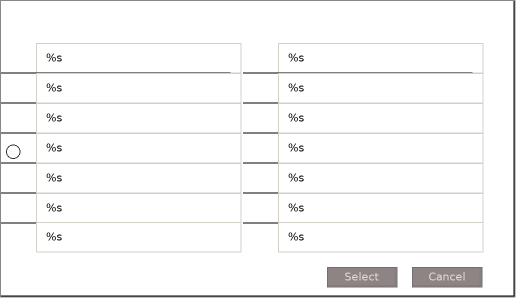
VISUALIZATION Visualization_FileList  // 516x298
    Rectangle (-1,0 515x296)
    Textfield (36,43 205x30), "%s", text variable: PRG_Process.arrFileNameList[1]
    Label (181,-2 158x39), "G-Code List"
    Line (230,73) (1,73)
    Line (230,103) (1,103)
    Line (230,133) (1,133)
    Line (230,163) (1,163)
    Line (230,193) (1,193)
    Line (230,223) (1,223)
    Textfield (36,73 205x30), "%s", text variable: PRG_Process.arrFileNameList[2]
    Textfield (36,103 205x30), "%s", text variable: PRG_Process.arrFileNameList[3]
    Textfield (36,133 205x30), "%s", text variable: PRG_Process.arrFileNameList[4]
    Textfield (36,163 205x30), "%s", text variable: PRG_Process.arrFileNameList[5]
    Textfield (36,193 205x30), "%s", text variable: PRG_Process.arrFileNameList[6]
    Textfield (36,222 205x30), "%s", text variable: PRG_Process.arrFileNameList[7]
    Textfield (278,43 205x30), "%s", text variable: PRG_Process.arrFileNameList[8]
    Line (472,73) (243,73)
    Line (472,103) (243,103)
    Line (472,133) (243,133)
    Line (472,163) (243,163)
    Line (472,193) (243,193)
    Line (472,223) (243,223)
    Textfield (278,73 205x30), "%s", text variable: PRG_Process.arrFileNameList[9]
    Textfield (278,103 205x30), "%s", text variable: PRG_Process.arrFileNameList[10]
    Textfield (278,133 205x30), "%s", text variable: PRG_Process.arrFileNameList[11]
    Textfield (278,163 205x30), "%s", text variable: PRG_Process.arrFileNameList[12]
    Textfield (278,193 205x30), "%s", text variable: PRG_Process.arrFileNameList[13]
    Textfield (278,222 205x30), "%s", text variable: PRG_Process.arrFileNameList[14]
    RadioButton (4,43 488x217), variable: PRG_Process.nFileNameList
    Button (327,267 70x20), "Select"
        tap PRG_Process.bSelectFile
    Button (412,267 70x20), "Cancel"
        tap PRG_Process.bCancelSelectFile
END_VISUALIZATION

(* stored: Version 1.1.0.1, ProductVersion 3.1.4022.6
   Visu Visualization_FileList: Id {495a280f-e8ae-4be7-be91-551c2c89de99} *)
